// TIA Portal project "Soru4" (V15)

(* hardware
DEVICE "S7-1200 station_1"  S7-1200 Station
   slot 0: "Rack_0"  S7-1200 Rack  Rack  V1.0
   slot 1: "PLC_1"  CPU 1214C DC/DC/DC  6ES7 214-1AG40-0XB0  V4.2
*)

// ===== PLC "PLC_1"  CPU 1214C DC/DC/DC =====

VAR_GLOBAL   // PLC tag table "Default tag table"
   "Dur" AT %I0.0 : Bool;
   "Basla" AT %I0.1 : Bool;
   "Motor_1" AT %Q0.0 : Bool;
   "Motor_2" AT %Q0.1 : Bool;
   "Motor_3" AT %Q0.2 : Bool;
   "Derğer" AT %MD0 : DWord;
END_VAR

// folder: System blocks/Program resources

DATA_BLOCK "Say"   // DB1
{ S7_Optimized_Access := 'TRUE' }
AUTHOR : Simatic
FAMILY : IEC
NAME : UCNTR
VERSION : 1.2
// stored: InstanceOfName IEC_UCOUNTER
"IEC_UCOUNTER"
BEGIN
END_DATA_BLOCK

// folder: (top level)

ORGANIZATION_BLOCK "Main"   // OB1, LAD, ProgramCycle
TITLE = "Main Program Sweep (Cycle)"
{ S7_Optimized_Access := 'TRUE' }
VERSION : 0.1
   VAR_INPUT
      Initial_Call : Bool;   // Initial call of this OB
      Remanence : Bool;   // =True, if remanent data are available
   END_VAR
BEGIN

REGION Network 1: Sayac ayarları
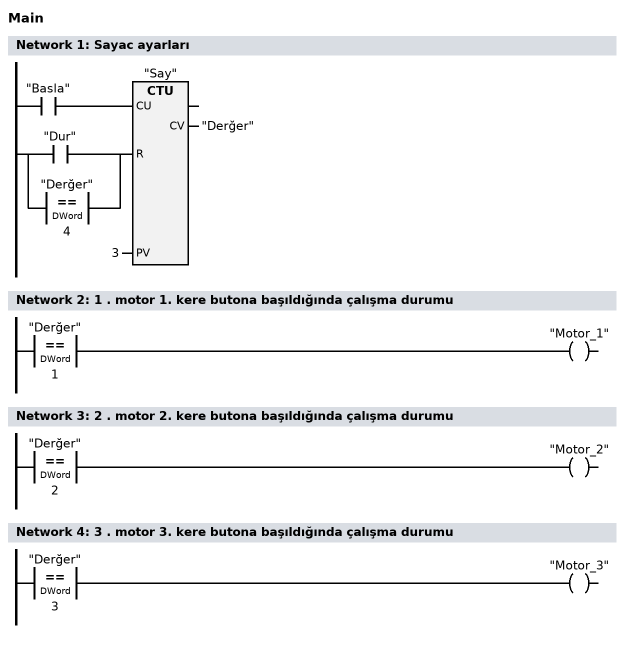
   "Say".CTU(CU := "Basla", R := "Dur" OR ("Derğer" = 4), PV := 3, CV => "Derğer");
END_REGION

REGION Network 2: 1 . motor 1. kere butona başıldığında çalışma durumu
   RUNG wire#powerrail
      { S7_Templates := "SrcType := DWord" } EQ_Contact(in1 := "Derğer", in2 := 1)
      Coil( "Motor_1" )
   END_RUNG
   // the same network as SCL:
   "Motor_1" := "Derğer" = 1;
END_REGION

REGION Network 3: 2 . motor 2. kere butona başıldığında çalışma durumu
   RUNG wire#powerrail
      { S7_Templates := "SrcType := DWord" } EQ_Contact(in1 := "Derğer", in2 := 2)
      Coil( "Motor_2" )
   END_RUNG
   // the same network as SCL:
   "Motor_2" := "Derğer" = 2;
END_REGION

REGION Network 4: 3 . motor 3. kere butona başıldığında çalışma durumu
   RUNG wire#powerrail
      { S7_Templates := "SrcType := DWord" } EQ_Contact(in1 := "Derğer", in2 := 3)
      Coil( "Motor_3" )
   END_RUNG
   // the same network as SCL:
   "Motor_3" := "Derğer" = 3;
END_REGION
END_ORGANIZATION_BLOCK